DATA_BLOCK "ST10_PMCountCycleTime"
VAR
  PM : Array[1..30] of "RCS_CountCycleTime_V1";
  PM_Num : Int;
END_VAR
BEGIN
END_DATA_BLOCK
